Universal Robots PolyScope program: Put_into_box_UR20.urp

Program Put_into_box_G6_UR20 (installation=default createdIn=3.0.0.0 lastSavedIn=5.10.0.1122333)
Robot Program (runOnlyOnce=true)
  Set NoAction (payload=0 tcpAsCog=true)
  MoveJ speed 50 deg/s, acceleration 100 deg/s^2 (useActiveTCP=false positionType=JointAngles) feature=Base
    Waypoint Home: TCP in base x=1.762 y=-291.18 z=1177.453 mm, rx=-0.0057 ry=2.2187 rz=-2.2189 rad; joints [0.001, -90.001, 0, -89.999, -0.001, 0.001] deg
    Waypoint End: TCP in base x=167.625 y=220.409 z=211.314 mm, rx=-2.0611 ry=-0.5234 rz=-2.1158 rad; joints [110, -190, 169.5, 102, 0, 0] deg
